# EPICS autosave request: iocBoot/iocStdVXTest/auto_settings.req
file "scan_settings.req",P=stdTest:,S=scan1
file "scan_settings.req",P=stdTest:,S=scan2
file "scan_settings.req",P=stdTest:,S=scan3
file "scan_settings.req",P=stdTest:,S=scan4

#file "femto.req",P=stdTest:,H=fem01:,F=seq01:
